Staubli VAL3: GetActionData.pgx

public program GetActionData(num& x_nSource[] (dimensions=3), num& x_nDest[] (dimensions=2), num x_nIndex)
  local num l_nX
  local num l_nY
begin

  //  x_nIndex=TxtFile:trCut[min(x_nIndex,size(TxtFile:pCut)-1)].y
  x_nIndex=roundDown(x_nIndex)
  if x_nIndex<=0 or x_nIndex>51
    //2014.4.10来实现
    //    for l_nX=0 to 11
    //      for l_nY=0 to 1
    //        x_nDest[l_nX,l_nY]=0
    //      endFor
    //    endFor
    x_nDest[0,0]=x_nDest[0,1]=x_nDest[1,0]=x_nDest[1,1]=x_nDest[2,0]=x_nDest[2,1]=x_nDest[3,0]=x_nDest[3,1]=0
    x_nDest[4,0]=x_nDest[4,1]=x_nDest[5,0]=x_nDest[5,1]=x_nDest[6,0]=x_nDest[6,1]=x_nDest[7,0]=x_nDest[7,1]=0
    x_nDest[8,0]=x_nDest[8,1]=x_nDest[9,0]=x_nDest[9,1]=x_nDest[10,0]=x_nDest[10,1]=x_nDest[11,0]=x_nDest[11,1]=0
    return
  endIf

  for l_nX=0 to 11
    for l_nY=0 to 1
      x_nDest[l_nX,l_nY]=x_nSource[x_nIndex,l_nX,l_nY]

    endFor
  endFor

end
